PROGRAM MAIN
VAR
END_VAR

Alias();
Permissives();
ChargeTime();
AnalogConversion();
VoltageMonitor();
Sequence();
HMI();
Heartbeat();

END_PROGRAM

(* stored: Version 1.1.0.1, ProductVersion 3.1.4024.11
   POU MAIN: Id {975ec784-f55e-4f2c-81eb-efc062cbd761}, SpecialFunc None *)
